{attribute 'GeneratedUsingTerminal: EL9520-0000-0016'}
{attribute addProperty BoxType "EL9520-0000-0016"}
{attribute addProperty Id "PowerOKAT %I*PowerOK_CEB2FD121WcStateAT %I*WcState_9091E0EB2InfoDataAT %I*InfoData_6F19DB2B2"}
{attribute addProperty CRC "3234029544"}
{attribute addProperty Size "5"}
TYPE EL9520_C0C35FE8 EXTENDS EtcSlaveTerminalBase_947E5A46 :
STRUCT
	{attribute addProperty Name "PowerOK"}
	PowerOK : PowerOK_CEB2FD12;
	{attribute addProperty Name "WcState"}
	WcState : WcState_9091E0EB;
	{attribute addProperty Name "InfoData"}
	InfoData : InfoData_6F19DB2B;
END_STRUCT
END_TYPE

(* stored: Version 1.2.0.0, ProductVersion 3.1.4024.9
   DUT EL9520_C0C35FE8: Id {b604888b-e3d3-471c-903f-9c188c745b3e} *)
